FUNCTION_BLOCK FB_RS_485
VAR
	Execute: BOOL;
	SendTimer: TON;
	fbTx :FB_FrameFifo;
	fbRx :FB_FrameFifo;(* Rx fifo *)
	SendErrorCount: INT;
	sSendData: STRING;
	sFromServer: STRING;
	
	fbsend:SendString;
	fbReceive: ReceiveString;
	
	bSendBusy:BOOL;
	Send_Error_ID:INT;
	Message: STRING;
	
	eState:E_ComState;
	ResponseTon: TON;
	SendMessageIndex: INT;
END_VAR

IF Execute THEN
	
	SendTimer( IN := TRUE, PT := GVL_CONSTANT.MFC_SEND_CYCLE_TIME);
	
	IF sendtimer.Q THEN
  		IF  fbtx.nCount < 5 THEN
			SendTimer( IN := FALSE);
			SendErrorCount:=0;
			
			_Make_Message();
		ELSE
			SendErrorCount :=  SendErrorCount+1;
			IF SendErrorCount > 10 THEN
				
				SendErrorCount:=0;
				fbtx.Clear();
				
			END_IF
		END_IF
	END_IF
	
	_Send_Received_Seq();
	
ELSE
	SendTimer( IN := FALSE);
	fbtx.Clear();
END_IF

REPEAT
	fbRx.RemoveHead();(* Fetch string from rx fifo *)
	IF fbRx.bOk THEN(* Success *)
		sFromServer := fbRx.sGet;
	END_IF
UNTIL NOT fbRx.bOk
END_REPEAT

ACTION _Make_Message:
//"@ADR" + STX + "RFV" + ETX + BCC
SendMessageIndex :=  SendMessageIndex +1;

CASE SendMessageIndex OF
	0:
		sSendData := F_BuildFrame(
END_CASE


IF sSendData <> '' THEN
	fbTx.AddTail(sPut:=sSendData);
END_IF
END_ACTION

ACTION _Received_Message:
////	Receive string data:
////	The block receives any data strings beginning with a STX ($02) and ending with an ETX ($03) character.
//TimeWaitReceive(IN := bSendingOK, PT := T#250MS); //Wait receiving data
//IF TimeWaitReceive.Q THEN
//	TimeWaitReceive(IN:= FALSE);
//	fbReceive(
//		Prefix:= '$02',
//		Suffix:= '$03',
//		Timeout:= T#1S,
//		ReceivedString:= sReceivedString,
//		RXbuffer:= GVL_Serial.RxBufferTB,
//		StringReceived=> bStringReceived,
//		Busy=> bReceiveBusy,
//		Error=> ,
//		RxTimeout=> bReceiveTimeout );
		
//	IF bReceiveTimeout THEN
//		isBath_Err[nReceivedBathNumber] := TRUE;
//		bReceiveTimeout := FALSE;
//	END_IF
	
//	IF fbReceive.Error <> COMERROR_NOERROR THEN
//		eReceiveErrorID := fbReceive.Error;
//	END_IF
	
//	IF bStringReceived THEN
//		bStringReceived :=FALSE;
//		bReceivedOK := TRUE;
//		bSendingEnable := TRUE;
//		sReceivedBathNumber := MID(STR:=sReceivedString, len:=1, pos:=3); //ReceivedString : '$0201$06PV100250$03'
//		nReceivedBathNumber := STRING_TO_INT(sReceivedBathNumber);
//		sReceivedAffirmation := MID(STR:=sReceivedString, len:=1, pos:=4); //Affirmation
		
//		IF bSetValueMode THEN //Write SV Mode
//			IF sReceivedAffirmation = '$06' THEN //'$06' ReceivedString : '$0201$06$03'
//				isBath_Err[nReceivedBathNumber] := FALSE;
//			ELSE
//				//isBath_Err[nReceivedBathNumber] := TRUE;
//			END_IF
//			bSetValueMode := FALSE;
//		ELSE //Read PV Mode
//			sReceivedData := MID(STR:=sReceivedString, len:=5, pos:=8); //ReceivedString : '$0201$06PV100250$03'
//			IF sReceivedData = '' THEN
//				isBath_Err[nReceivedBathNumber] := TRUE;
//				;
//			ELSIF sReceivedData = 'HHHHH' THEN
//				rTemperature_PV[nReceivedBathNumber] := -99.0;
//				isBath_TC_Broken[nReceivedBathNumber] := TRUE;
//				isBath_Err[nReceivedBathNumber] := FALSE;
//			ELSE
//				rTemperature_PV[nReceivedBathNumber] := (STRING_TO_REAL(sReceivedData))/10;
//				isBath_TC_Broken[nReceivedBathNumber] := FALSE;
//				isBath_Err[nReceivedBathNumber] := FALSE;
//			END_IF
//		END_IF
//	END_IF
	
	

//	bSendingEnable := TRUE;
//END_IF
END_ACTION

ACTION _Send_Received_Seq:

CASE eState OF
	E_ComState.IDLE:
		Message:='Wait Message';
		IF fbTx.nCount > 0 THEN
			eState := E_ComState.OPEN;
		END_IF
		
	E_ComState.OPEN:
		eState := E_ComState.CONNECTED;
		
	E_ComState.CONNECTED:
		eState := E_ComState.SENDING;
		
		
	E_ComState.EXIST_MSG:
		IF fbTx.nCount > 0 THEN
			fbTx.RemoveHead( sGet => sSendData );
			IF fbTx.bOk THEN(* Success *)
				eState := E_ComState.SENDING;
			END_IF
		ELSE
			eState:=E_ComState.IDLE;
		END_IF
		

	E_ComState.SENDING:
		IF fbsend.Busy = FALSE AND LEN(sSendData) > 2 THEN
			fbSend(	
				SendString:= sSendData,
				TXbuffer:= GVL_Serial.TxBufferTB_MFC,
				Busy=> bSendBusy,
				Error=>);
			
			IF fbSend.Error <> COMERROR_NOERROR THEN
				Send_Error_ID := fbSend.Error;
				eState:=E_ComState.CLOSING;
			ELSE
				Send_Error_ID := COMERROR_NOERROR;
				eState:=E_ComState.WAITING_RESPONSE;
			END_IF
		END_IF
	
	E_ComState.WAITING_RESPONSE:
		ResponseTon(IN:=TRUE,PT:=T#200MS);
			IF ResponseTon.Q THEN
				ResponseTon(IN:= FALSE);
				IF fbReceive.Busy = FALSE THEN
					fbReceive(
						Prefix:= '$02',
						Suffix:= '$03',
						Timeout:= T#1S,
						ReceivedString:= sFromServer,
						RXbuffer:= GVL_Serial.RxBufferTB_MFC,
						StringReceived=>,
						Busy=> ,
						Error=> ,
						RxTimeout=>  );
						
						eState:=E_ComState.PARSING;
				END_IF
			END_IF
			
		E_ComState.PARSING:
		;
		
		
END_CASE
END_ACTION

END_FUNCTION_BLOCK

(* stored: Version 1.1.0.1, ProductVersion 3.1.4024.15
   POU FB_RS_485: Id {32fd6766-f533-4360-b206-acf29707e36e}, SpecialFunc None
   Action _Make_Message: Id {be4cbf91-f7eb-443c-ac3e-5bf2fab3f002}
   Action _Received_Message: Id {18298bf7-a05f-4afc-ac68-91cedbab7e99}
   Action _Send_Received_Seq: Id {bf670ca1-3e9d-40bd-a1d1-9147e676c0af} *)
